{attribute 'qualified_only'}
VAR_GLOBAL
	bXAxisEnable : BOOL;
	
	
END_VAR

(* stored: Version 1.1.0.1, ProductVersion 3.1.4024.3
   GVL GVL_AxisCtr: Id {b11b1f42-c440-4ccb-b90d-2c1361b57084} *)
